// TIA Portal V19 export
TYPE "C215_STU_IF_DVLU_TYPIC"
   STRUCT
      CMD_OPL { ExternalAccessible := 'False'; ExternalVisible := 'False'; ExternalWritable := 'False'} : Bool;   // Aansturing indicatiebord vluchtroute oplopende richting
      CMD_AFL { ExternalAccessible := 'False'; ExternalVisible := 'False'; ExternalWritable := 'False'} : Bool;   // Aansturing indicatiebord vluchtroute aflopende richting
      CMD_RES { ExternalAccessible := 'False'; ExternalVisible := 'False'; ExternalWritable := 'False'} : Bool;   // Reset van de latched storingen
   END_STRUCT;
END_TYPE
